// TwinCAT 3 PLC project VFD_Control
// ProgramVersion: 3.1.4023.0
// libraries:
//   Tc2_Standard, * (Beckhoff Automation GmbH)
//   Tc2_System, * (Beckhoff Automation GmbH)
//   Tc3_Module, * (Beckhoff Automation GmbH)
// project tree:
//   DUTs/ eControlModeVent.TcDUT
//   / PlcTask.TcTTO
//   POUs/ FB_RetrieveLowerLimit.TcPOU, FB_UpperLimitRetrieval.TcPOU, FB_VentilationControl.TcPOU, MAIN.TcPOU
// real-time tasks:
//   TASK PlcTask: cycle T#10ms, priority 20, ADS port 350

CONFIGURATION VFD_Control
    RESOURCE PLC ON TwinCAT3
        TASK PlcTask(INTERVAL := T#10ms, PRIORITY := 20);
        PROGRAM MAIN WITH PlcTask : MAIN;
    END_RESOURCE
END_CONFIGURATION

// ---- DUTs/eControlModeVent.TcDUT
{attribute 'qualified_only'}
{attribute 'strict'}
TYPE eControlModeVent :
(
	Normal := 0,
	Adapted := 1,
	NewRegime := 2
);
END_TYPE

// ---- POUs/MAIN.TcPOU
PROGRAM MAIN
VAR
END_VAR

END_PROGRAM

// ---- POUs/FB_RetrieveLowerLimit.TcPOU
FUNCTION_BLOCK FB_RetrieveLowerLimit
VAR_INPUT
	bCooling : BOOL;
    fTfruitHot : REAL; // Fruit temperature sensor at hot side of the room
    fTfruitCold : REAL; // fruit temperature sensor at cold side of the room
    bUpdateRequested : BOOL;
END_VAR
VAR_OUTPUT
	bRetrievingLowerLimit : BOOL;
    bLowerLimitRetrieved : BOOL := FALSE;
    fCurrentLowerLimit : REAL :=999.99; //If fCurrentUpperLimit = 999.99 then we know that it isn't set yet 
END_VAR
VAR
	fStartDiff_lowerlimit : REAL;
    fEndDiff_lowerlimit : REAL;
    fMax_lowerlimit : REAL;
    tTimeForVentilation : TIME := T#20M; // 20 minutes
    timer : TON;
    bTimer_done : BOOL;
    bStartVentilating : BOOL; // Boolean to start the ventilation process
END_VAR

R_trig(CLK:=bUpdateRequested);
IF R_trig.Q AND NOT bRetrievingLowerLimit THEN
	bRetrievingLowerLimit := TRUE;
	bLowerLimitRetrieved := FALSE;
END_IF

IF bRetrievingLowerLimit THEN
	F_trig(CLK := bCooling);
END_IF

IF (F_trig.Q) AND bRetrievingLowerLimit THEN // falling edge --> faling edge bCooling
	bStartVentilating := TRUE; // Signal to start the ventilation process
	fStartDiff_lowerlimit := ABS(fTfruitHot - fTfruitCold);
END_IF

IF bStartVentilating AND bRetrievingLowerLimit THEN
	timer(IN := bStartVentilating, PT := tTimeForVentilation, Q => bTimer_done); // wait for 20 minutes
	IF bTimer_done THEN
		fEndDiff_lowerlimit := ABS(fTfruitHot - fTfruitCold);
		fMax_lowerlimit := fStartDiff_lowerlimit - fEndDiff_lowerlimit;
		bStartVentilating := False;
		bLowerLimitRetrieved := TRUE;
		bRetrievingLowerLimit := FALSE;
	END_IF
END_IF

fCurrentLowerLimit := fMax_lowerlimit;

END_FUNCTION_BLOCK

// ---- POUs/FB_UpperLimitRetrieval.TcPOU
FUNCTION_BLOCK FB_UpperLimitRetrieval
VAR_INPUT
    bStartDCA : BOOL;
    bUpdateRequested : BOOL;
    fTfruitHot : REAL; // fruit temperature at hot side of the room
    fTfruitCold : REAL; // fruit temperature at cold side of the room
END_VAR
VAR_OUTPUT
    fLatestUpperLimit : REAL ;
	fCurrentUpperLimit : REAL := 999.99; //If fCurrentUpperLimit = 999.99 then we know that it isn't set yet
END_VAR
VAR
	bDcaStarted : BOOL := FALSE;
    fStartDiff_upperlimit : REAL;
    fEndDiff_upperlimit : REAL;
    fMax_upperlimit : REAL;
    tTimeForUpperLimitLog : TIME := T#30M;
    bTimer_done : BOOL;
	timer : TON;
END_VAR

R_trig(CLK:=bStartDCA);
IF R_trig.Q THEN // positive edge trigger of a DCA action
	bDcaStarted:= TRUE;
END_IF

IF bDcaStarted THEN
    fStartDiff_upperlimit := ABS(fTfruitHot - fTfruitCold);
    timer(IN := bDcaStarted, PT := tTimeForUpperLimitLog, Q => bTimer_done); // wait for 20 minutes
    IF bTimer_done THEN
        fEndDiff_upperlimit := ABS(fTfruitHot - fTfruitCold);
        fMax_upperlimit := fStartDiff_upperlimit - fEndDiff_upperlimit;
        fLatestUpperLimit := fMax_upperlimit;
		bDcaStarted := FALSE;
    END_IF
END_IF

IF bUpdateRequested THEN
    fCurrentUpperLimit := fLatestUpperLimit;
END_IF

END_FUNCTION_BLOCK

// ---- POUs/FB_VentilationControl.TcPOU
FUNCTION_BLOCK FB_VentilationControl
VAR_INPUT
	fTfruitHot : REAL; // Fruit temperature sensor at hot side of the room
    fTfruitCold : REAL; // Fruit temperature sensor at cold side of the room
    bVent20: BOOL;          // Digital input connected to 39K1 relay for 20 % ventilation which is connected to LI1
    bVent80: BOOL;         // Digital input connected to 39K3 relay for 80 % ventilation which is connected to LI2
    bCooling: BOOL;         // Digital input connected to valve relay of the cooling liquid
    bScrubbing: BOOL;       // Digital input conncted to ectronic relay of the motor for scrubbing
    eControlModeVent : eControlModeVent; // control mode input
    bStartDCA: BOOL;              // A boolean that is true if a DCA action starts
    bResetControl: BOOL;     // Reset mode
    bUpdateLimits: BOOL;    // To update the recommended limit values
END_VAR
VAR_OUTPUT
	bVent100Control: BOOL;   // Digital output connected to relay K1 which will be connected to LI3
    bVentZeroControl: BOOL;   // Digital output connected to relay K2 which will be connected to LI4
    fCurrentMode: LREAL;     // To display the current control mode
    fLatestUpperLimit : REAL := 999;
END_VAR
VAR
    Retrieving_lowerLimit : FB_RetrieveLowerLimit;
	Retrieving_upperLimit : FB_UpperLimitRetrieval;
	bRetrieving_lowerlimit : BOOL;
    bLowerLimitRetrieved : BOOL;
	bUpdateRequested : BOOL;
	bCoolingJustEnded : BOOL;
END_VAR
VAR_IN_OUT
    fUpperLimit : REAL := 0.0; // Input of the upper limit done by the grower, based on the recommended limit
    fLowerLimit : REAL := 0.0; // Input of the lower limit done by the grower, based on the recommended limit
END_VAR

R_trig(CLK:=bUpdateLimits);
IF R_trig.Q THEN // this will trigger an update request for the lower limit. And it will update the upper limit to the latest value.
    bUpdateRequested := TRUE;
END_IF

IF bUpdateRequested THEN
Retrieving_upperLimit(bStartDCA := bStartDCA,
                    bUpdateRequested := bUpdateRequested,
                    fTfruitHot := fTfruitHot,
                    fTfruitCold := fTfruitHot,
                    fCurrentUpperLimit => fUpperLimit,
                    fLatestUpperLimit => fLatestUpperLimit);

Retrieving_lowerLimit(bCooling := bCooling,
                    bUpdateRequested := bUpdateRequested,
                    fTfruitHot := fTfruitHot,
                    fTfruitCold := fTfruitCold,
                    fCurrentLowerLimit => fLowerLimit,  
                    bRetrievingLowerLimit => bRetrieving_lowerlimit,
                    bLowerLimitRetrieved => bLowerLimitRetrieved);
    IF bLowerLimitRetrieved THEN // Reset the request boolean, UpperLimit is always "Up to date"
        bUpdateRequested := FALSE;
    END_IF	
END_IF

//////////////////////////////Mode control////////////////////////////////////////////////////////////////////////

IF (eControlModeVent = 0) THEN // normal regime mode (all at 50 Hz)
    fCurrentMode := eControlModeVent;
    bVent100Control := TRUE;
END_IF

IF (eControlModeVent = 1) THEN // adapted regime mode (rest ventilation at 40 Hz)
    fCurrentMode := eControlModeVent;
    IF (bVent20 AND bVent80 AND bCooling) THEN
        bVent100Control := TRUE; // sets the ventilation from 80 % to 100 % during cooling actions
    //Else: do nothing and leave the ventilation at 80 % --> everey action is 80 % unless tge 
    END_IF
END_IF

IF (eControlModeVent = 2) THEN // newly proposed regime mode (rest ventilation based on warm and cold temperature)
	F_trig(CLK := bCooling);
	IF F_trig.Q THEN
		bCoolingJustEnded := TRUE;
	END_IF
	IF bCooling THEN
		bCoolingJustEnded := FALSE;
		bVent100Control := TRUE;
	END_IF
	
    IF (bCoolingJustEnded AND NOT bScrubbing) THEN //Rest ventilation
        bVentZeroControl := TRUE; // sets the ventilation at 0 % between cooling actions, but not during scrubbing actions
        IF (ABS(fTfruitHot - fTfruitCold) >= fUpperLimit) THEN // above the upper limit, the vetilation should be ON (unless a scrubber action or defrosting actions will take place)
            bVentZeroControl := FALSE; //ventilating op 80 %
        // activating bVent20 and bVent80
        ELSIF ((ABS(fTfruitHot - fTfruitCold) < fLowerLimit)) THEN
            bVentZeroControl := TRUE;
			bVent100Control := TRUE;
        END_IF
	ELSIF (bRetrieving_lowerlimit) THEN
        bVent100Control := TRUE;
	ELSIF bScrubbing THEN
		bVentZeroControl := FALSE;
    END_IF
END_IF
    IF (bRetrieving_lowerlimit) THEN
        bVent100Control := TRUE;
END_IF

END_FUNCTION_BLOCK
